{attribute 'qualified_only'}
VAR_GLOBAL INTERNAL
	stDebug				: ARRAY[0..Param.nMaxDebugArraySize] OF ST_DebugInfo;
	nDebugLen			: UDINT;	
END_VAR

(* stored: Version 1.1.0.1
   GVL _Debug: Id {2a504fcf-83e8-4dbb-bb0d-d2a7e0a5f5bb} *)
